Omron CX-Programmer project NewProject (CX-Programmer 9.51)

# PLC my_first_project: CP1L L
; comment

## Global symbols (name address type ; comment)
0.00 BOOL  ; commnt
0.01 BOOL  ; comment
100.00 BOOL  ; comment
100.01 BOOL  ; comment

## Program NewProgram1 (cyclic task 0)
Local symbols
button_1 0.00 BOOL  ; comment
button_2 0.01 BOOL  ; Comment
button_3 0.02 BOOL  ; Comment
out_1 100.00 BOOL  ; comment
out_2 100.01 BOOL  ; comment
out_3 100.02 BOOL  ; comment

### Section Section1

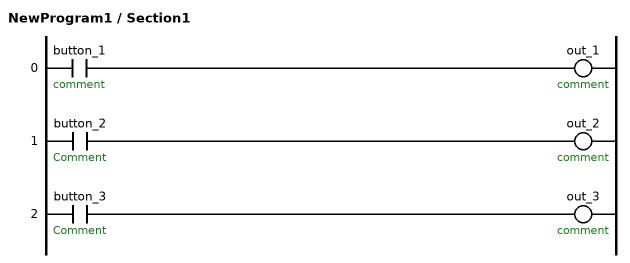
; rung 0
LD button_1  ; comment
OUT out_1  ; comment
; rung 1
LD button_2  ; Comment
OUT out_2  ; comment
; rung 2
LD button_3  ; Comment
OUT out_3  ; comment

### Section END
; rung 0
END(001)